TYPE ST_MinMax :
STRUCT
	mini : REAL;
	maxi : REAL;
END_STRUCT
END_TYPE

(* stored: Version 1.1.0.1, ProductVersion 3.1.4024.16
   DUT ST_MinMax: Id {dc5be70b-cb0e-4224-8cf5-e642e31760a6} *)
